TYPE Station001_ProductionData EXTENDS TcoData.TcoEntity:
STRUCT
	Result : BOOL;
	RecipeName : STRING;
	DimX : AnalogueValueCheck;
	DimY : AnalogueValueCheck;
	DimZ : AnalogueValueCheck;
END_STRUCT
END_TYPE

(* stored: Version 1.1.0.1, ProductVersion 3.1.4024.9
   DUT Station001_ProductionData: Id {148e1532-fd36-4606-a278-36ddc44c44a7} *)
